# B&R Automation Studio project SFL4_Manitou_230503
Automation Studio 4.9

## Configuration Config1

### Hardware
```
X90CP174_24_00 : X90CP174.24-00 v1.3.1.0  [X1 -> X1.SL]
  Module X1 (Type=X1, Virtual=true, Version=1.3.1.0)
    Connection (Connector=SL, TargetModule=X90CP174_24_00, TargetConnector=X1)
  Connector IF2:
    ActivateDevice = 1
  ConfigurationID = SFL4_Manitou_230503_Config1
  Cyclic1Duration = 10000
  Cyclic1Tolerance = 10000
  Cyclic2Duration = 20000
  Cyclic2Tolerance = 20000
  Cyclic3Duration = 50000
  Cyclic3Tolerance = 50000
  Cyclic4Duration = 100000
  Cyclic4Tolerance = 100000
  Cyclic5Duration = 200000
  Cyclic5Tolerance = 200000
  Cyclic6Duration = 500000
  Cyclic6Tolerance = 500000
  Cyclic7Duration = 1000000
  Cyclic7Tolerance = 1000000
  Cyclic8Duration = 10000
  Cyclic8Tolerance = 30000000
```

### Config.mpdatabasecore - X90CP174_24_00/mappServices/Config.mpdatabasecore
```
Element gDatabaseCore (Type=mpdatabasecore)
  mapp.Database.Core:
    Name = manitou
    UserName = Manitou
    Password = Ganz_Wien79
    IPAddress = 10.16.2.233
    PortNumber = 3306
```

## Logical view

Binary libraries used (declarations not repeated): operator, runtime, astime, AsIecCon, MpDatabase, MpBase, AsHttp

### Program Logical/Program

#### Variables.var
```iecst
VAR
	MpDatabaseCore_0 : MpDatabaseCore;
END_VAR
```

#### Cyclic.ld
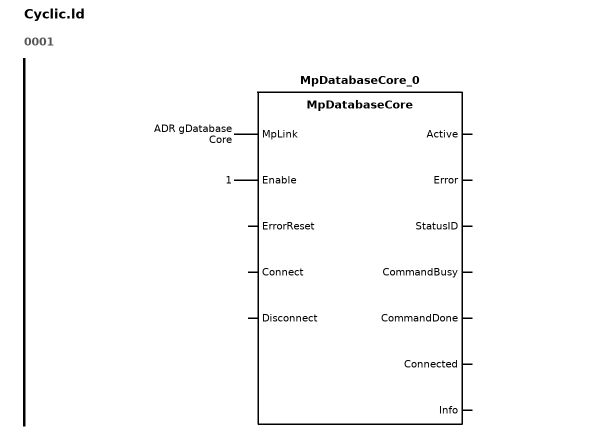
Ladder, written as Structured Text:
```iecst
PROGRAM _CYCLIC
(* Network 1 *)
MpDatabaseCore_0(MpLink := ADR(gDatabaseCore), Enable := 1);
END_PROGRAM
```

#### Exit.ld
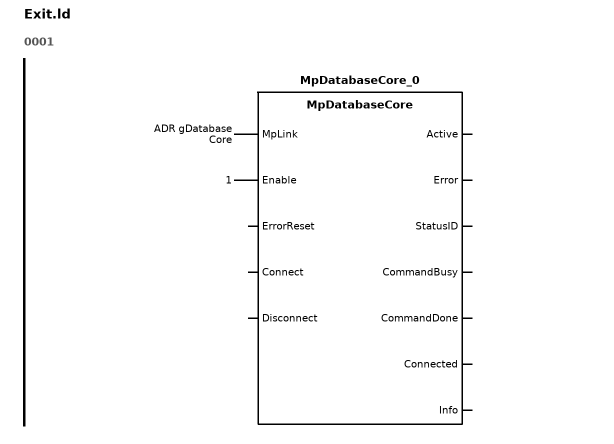
Ladder, written as Structured Text:
```iecst
PROGRAM _EXIT
(* Network 1 *)
MpDatabaseCore_0(MpLink := ADR(gDatabaseCore), Enable := 1);
END_PROGRAM
```

#### Init.ld
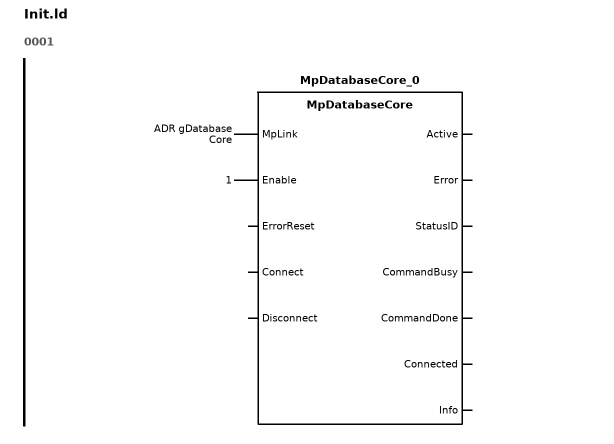
Ladder, written as Structured Text:
```iecst
PROGRAM _INIT
(* Network 1 *)
MpDatabaseCore_0(MpLink := ADR(gDatabaseCore), Enable := 1);
END_PROGRAM
```

Listed in the project but not available here: Logical/Libraries/ManProgram
